PROGRAM WateringTask
VAR
	WaterTimer:TON;
	Delay:TON;
	state:INT;
	Moisture: REAL;
	Temp: REAL;
	WaterRequired: BOOL;
END_VAR

 	
//Watering control
CASE state OF
	
	
	0:// Initial position
	gvl.WaterON:= FALSE;
	state:=1;
	1:// Checking the conditions
	IF gvl.WaterRequired THEN
				gvl.WaterDuration := GetWaterDuration(gvl.Moisture, Temp);
				gvl.WaterON := TRUE;	
				WaterTimer(IN := TRUE, PT := gvl.WaterDuration);
				State := 2;
			ELSE
				State := 3;
			END_IF;
			
	2:  // Watering
	WaterTimer(IN := TRUE);
			IF WaterTimer.Q THEN
			  gvl.WaterON := FALSE;
	GVL.WaterRequired := FALSE;
	END_IF
	WaterTimer(IN := FALSE);
				state := 3;
	3:// Idle
	Delay(IN:=TRUE, PT:=T#5S);
	IF NOT(Delay.Q) THEN
		RETURN;
	END_IF
	Delay(In:=FALSE);
	state:=1;		
END_CASE

END_PROGRAM

(* stored: Version 1.1.0.1, ProductVersion 3.1.4024.15
   POU WateringTask: Id {b5a1694e-819d-48dc-a239-eb210722768b}, SpecialFunc None *)
